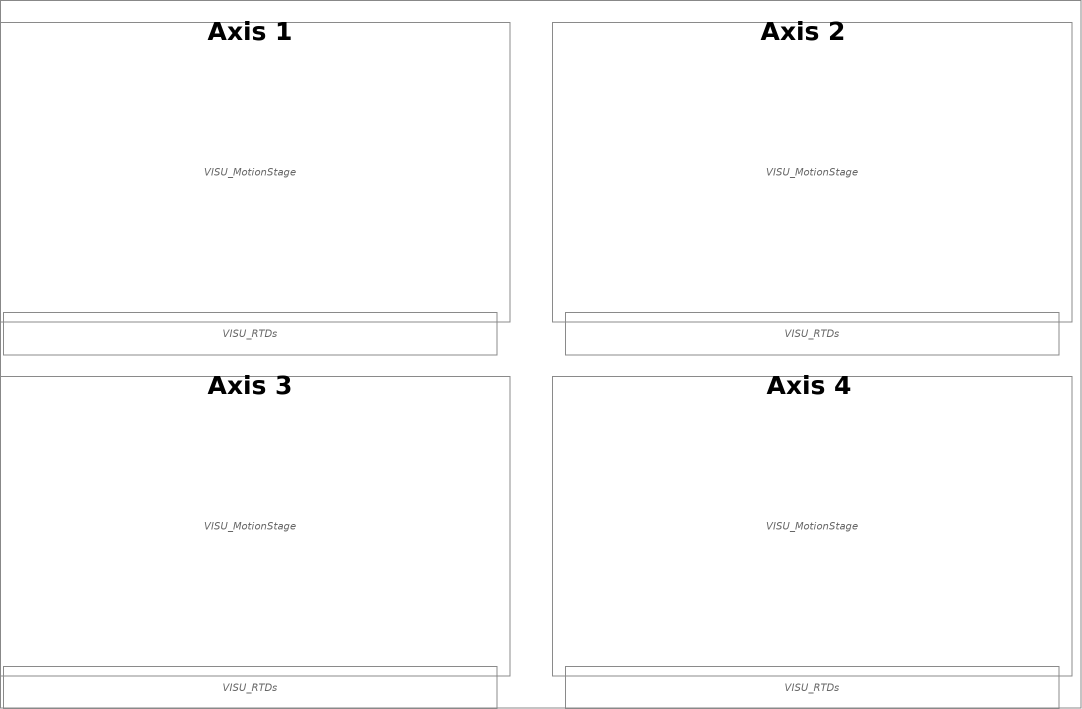
VISUALIZATION AT1K4  // 1082x709
    Frame (-10,22 520x300)
        shows VISU_MotionStage(VisuMotionStage := Main.M1, Extras := PRG_2_AT1K4.fbSATT.fbStage1.stExtra)
    Frame (3,312 494x43)
        shows VISU_RTDs(fTemp1 := PRG_2_AT1K4.fbSATT.RTD_Axis1_1.fTemp, fTemp2 := PRG_2_AT1K4.fbSATT.RTD_Axis1_2.fTemp)
    Label (82,15 336x32), "Axis 1"
    Frame (552,22 520x300)
        shows VISU_MotionStage(VisuMotionStage := Main.M2, Extras := PRG_2_AT1K4.fbSATT.fbStage2.stExtra)
    Frame (565,312 494x43)
        shows VISU_RTDs(fTemp1 := PRG_2_AT1K4.fbSATT.RTD_Axis2_1.fTemp, fTemp2 := PRG_2_AT1K4.fbSATT.RTD_Axis2_2.fTemp)
    Label (635,15 336x32), "Axis 2"
    Frame (-10,376 520x300)
        shows VISU_MotionStage(VisuMotionStage := Main.M3, Extras := PRG_2_AT1K4.fbSATT.fbStage3.stExtra)
    Frame (3,666 494x43)
        shows VISU_RTDs(fTemp1 := PRG_2_AT1K4.fbSATT.RTD_Axis3_1.fTemp, fTemp2 := PRG_2_AT1K4.fbSATT.RTD_Axis3_2.fTemp)
    Label (82,369 336x32), "Axis 3"
    Frame (552,376 520x300)
        shows VISU_MotionStage(VisuMotionStage := Main.M4, Extras := PRG_2_AT1K4.fbSATT.fbStage4.stExtra)
    Frame (565,666 494x43)
        shows VISU_RTDs(fTemp1 := PRG_2_AT1K4.fbSATT.RTD_Axis4_1.fTemp, fTemp2 := PRG_2_AT1K4.fbSATT.RTD_Axis4_2.fTemp)
    Label (641,369 336x32), "Axis 4"
END_VISUALIZATION

(* stored: Version 1.1.0.1, ProductVersion 3.1.4024.4
   Visu AT1K4: Id {b96f1ec7-b5de-4fc7-8dac-be4f07fb29e8} *)
